// TIA Portal V17 export
// export: Created 2022-12-08T10:17:02.5462407Z, ExportSetting WithDefaults, DisplayName Totally Integrated Automation Portal, DisplayVersion V17 Update 5, DisplayName TIA Portal Openness, DisplayVersion V17 Update 5, DisplayName TIA Portal Version Control Interface, DisplayVersion V17, DisplayName Simotion SCOUT TIA, DisplayVersion 5.4.3.0, DisplayName SINAMICS Startdrive Advanced, DisplayVersion V17 SP1, DisplayName SINAMICS Startdrive G130, G150, S120, S150, SINAMICS MV, S210, DisplayVersion V17 SP1, DisplayName SINAMICS Startdrive G110M, G120, G120C, G120D, G120P, G115D, DisplayVersion V17 SP1, DisplayName STEP 7 Professional, DisplayVersion V17 Update 5, DisplayName STEP 7 Safety, DisplayVersion V17, DisplayName WinCC Advanced, DisplayVersion V17 Update 5
DATA_BLOCK "DB_SIKO"   // DB16
VERSION : 0.1
// stored: AutoNumber true, DBAccessibleFromOPCUA true, DBAccessibleFromWebserver true, InstanceOfName FB_SIKO, InstanceOfType FB
"FB_SIKO"
   // VAR_INPUT
   //    i_nodes : Array[0..31] of HW_IO;
   //    i_enable : Bool;
   //    i_reset : Bool;
   //    i_NodeUp : Bool;
   //    i_NodeDown : Bool;
   //    i_CurrentPictureNumber : Int;
   //    i_PictureNumber : Int;
   //    i_UpperLimitNode : Int;
   // END_VAR
   // VAR_OUTPUT
   //    q_NodeNumbersNotInRange : String;
   //    q_AllNodesInRange : Bool;
   //    q_ActiveNodeNumber : Int;
   // END_VAR
   // VAR_IN_OUT
   //    iq_HMISIKO : "UDT_SIKO";
   //    iq_HMIData : "UDT_SIKODATA";
   //    iq_SIKO : Array[0..31] of "UDT_SIKO";
   //    iq_SIKOData : Array[0..31] of "UDT_SIKODATA";
   // END_VAR
   // VAR
   //    stat_FirstCycle : Bool;
   //    stat_NodeNumber : Int;
   //    stat_NodeNumberOld : Int;
   //    stat_NodeNumbersNotInRange : String;
   //    stat_TONEnable : TON_TIME;
   //    stat_RTRIGReadOnce : R_TRIG;
   //    stat_RTRIGNodeUp : R_TRIG;
   //    stat_RTRIGNodeDown { S7_SetPoint := 'True'} : R_TRIG;
   //    stat_SIKO_POS_AP10vPN { S7_SetPoint := 'True'} : Array[0..31] of "SIKO_POS_AP10vPN";
   // END_VAR
BEGIN
END_DATA_BLOCK
